// TIA Portal project "Factory_io_Analog_Assembler_with tia_portal_s7_plc1200_sequential" (V16)

(* hardware
DEVICE "S7-1200 station_1"  S7-1200 Station
   slot 0: "Rack_0"  S7-1200 Rack  Rack  V1.0
   slot 1: "PLC_1"  CPU 1212C DC/DC/Rly  6ES7 212-1HE40-0XB0  V4.4
   slot 2: "AI 4x16BIT_1"  SM 1231 AI4 x HF  6ES7 231-5ND32-0XB0  V2.0
   slot 3: "AQ 2x16BIT_1"  SM 1232 AQ2  6ES7 232-4HB32-0XB0  V2.1
*)

// ===== PLC "PLC_1"  CPU 1212C DC/DC/Rly =====

VAR_GLOBAL   // PLC tag table "Default tag table"
   "X_Current_Value" AT %ID1 : Real;
   "Z_Current_Value" AT %ID5 : Real;
   "Set_X" AT %QD30 : Real;
   "Set_Z" AT %QD34 : Real;
   "x scale for x" AT %MD44 : Real;
   "x rounded" AT %MD88 : Real;   // x rounded *10
   "Scale_X_For_Z" AT %MD48 : Real;
   "Z_rounded" AT %MD84 : Real;   // z rounded * 10
   "Item Detected" AT %I0.0 : Bool;
   "Lid At Place" AT %I0.1 : Bool;
   "Base At Place" AT %I0.2 : Bool;
   "Part Leaving" AT %I0.3 : Bool;
   "Start" AT %I0.4 : Bool;
   "Reset" AT %I0.5 : Bool;
   "Manual" AT %I0.6 : Bool;
   "auto" AT %I0.7 : Bool;
   "Lid Conveyor 1" AT %Q0.0 : Bool;
   "Stop Blade     1" AT %Q0.1 : Bool;
   "Lid Conveyor 2" AT %Q0.2 : Bool;
   "Base Conveyor 1" AT %Q0.3 : Bool;
   "Stop blad        2" AT %Q0.4 : Bool;
   "Base Conveyor 2" AT %Q0.5 : Bool;
   "Grab" AT %Q0.6 : Bool;
   "Start Light" AT %Q0.7 : Bool;
   "Memory for Postive edge of start" AT %M0.0 : Bool;
   "Start_FC_one_time" AT %M0.1 : Bool;
   "Cycle complete" AT %M0.2 : Bool;
   "Negative edge for lid conveyor 1" AT %M0.3 : Bool;
   "Negative edge for base conveyor 1" AT %M0.4 : Bool;
   "Negative edge for grab" AT %M0.5 : Bool;
   "Negative edge for Stop Blade 2" AT %M0.6 : Bool;
   "Postive edge for lid at place" AT %M0.7 : Bool;
   "Postive Edge For Base At Place" AT %M1.0 : Bool;
   "Negative edge for part leaving" AT %M1.1 : Bool;
   "postive edge for part leaving" AT %M1.2 : Bool;
   "finished product counter" AT %QD38 : DWord;
END_VAR

DATA_BLOCK "modes"   // DB1
{ S7_Optimized_Access := 'FALSE' }
VERSION : 0.1
   VAR
      "Reset Mode" : Bool;
      "Manual Mode" : Bool;
      "Auto Mode" : Bool;
   END_VAR
BEGIN
END_DATA_BLOCK

DATA_BLOCK "Step_Data"   // DB2
{ S7_Optimized_Access := 'TRUE' }
VERSION : 0.1
   VAR
      "Set X" : Real;
      "Set Z" : Real;
      "Lid Conveyor 1" : Bool;
      "Base Conveyor 1" : Bool;
      "Base Conveyor 2" : Bool;
      Grab : Bool;
      "Stop Blade 1" : Bool;
      "Stop Blade 2" : Bool;
      Every_thing_AT_home : Bool;
   END_VAR
BEGIN
END_DATA_BLOCK

DATA_BLOCK "Steps"   // DB3
{ S7_Optimized_Access := 'TRUE' }
VERSION : 0.1
   VAR
      Current_step : Int;
   END_VAR
BEGIN
END_DATA_BLOCK

// folder: System blocks/Program resources

DATA_BLOCK "IEC_Counter_0_DB"   // DB4
{ S7_Optimized_Access := 'TRUE' }
AUTHOR : Simatic
FAMILY : IEC
NAME : CNTR
VERSION : 1.0
// stored: InstanceOfName IEC_COUNTER
"IEC_COUNTER"
BEGIN
END_DATA_BLOCK

// folder: (top level)

FUNCTION "round_x and z" : Void   // FC1, LAD
{ S7_Optimized_Access := 'TRUE' }
VERSION : 0.1
BEGIN

REGION Network 1
   // Z rounded x10
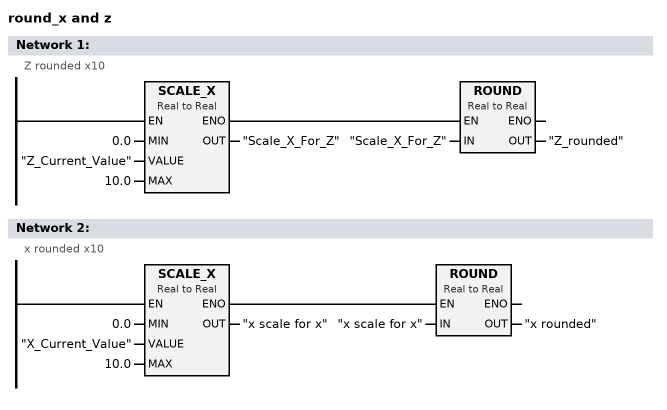
   RUNG wire#powerrail
      { S7_Templates := "[SrcType := Real, DestType := Real]" } Scale(min := 0.0, value := "Z_Current_Value", max := 10.0, out => "Scale_X_For_Z")
      { S7_Templates := "[SrcType := Real, DestType := Real]" } Round(in := "Scale_X_For_Z", out => "Z_rounded")
   END_RUNG
   // the same network as SCL:
   "Scale_X_For_Z" := SCALE_X(MIN := 0.0, VALUE := "Z_Current_Value", MAX := 10.0);
   "Z_rounded" := ROUND("Scale_X_For_Z");
END_REGION

REGION Network 2
   // x rounded x10
   RUNG wire#powerrail
      { S7_Templates := "[SrcType := Real, DestType := Real]" } Scale(min := 0.0, value := "X_Current_Value", max := 10.0, out => "x scale for x")
      { S7_Templates := "[SrcType := Real, DestType := Real]" } Round(in := "x scale for x", out => "x rounded")
   END_RUNG
   // the same network as SCL:
   "x scale for x" := SCALE_X(MIN := 0.0, VALUE := "X_Current_Value", MAX := 10.0);
   "x rounded" := ROUND("x scale for x");
END_REGION
END_FUNCTION

FUNCTION "Step_definition" : Void   // FC2, LAD
{ S7_Optimized_Access := 'TRUE' }
VERSION : 0.1
   VAR_TEMP   // added for the SCL form of the ladder/FBD networks
      _w1 : Bool;
   END_VAR
BEGIN

REGION Network 1: turn on lid conveyor till lid at place
   // start pressed  and every thing at home
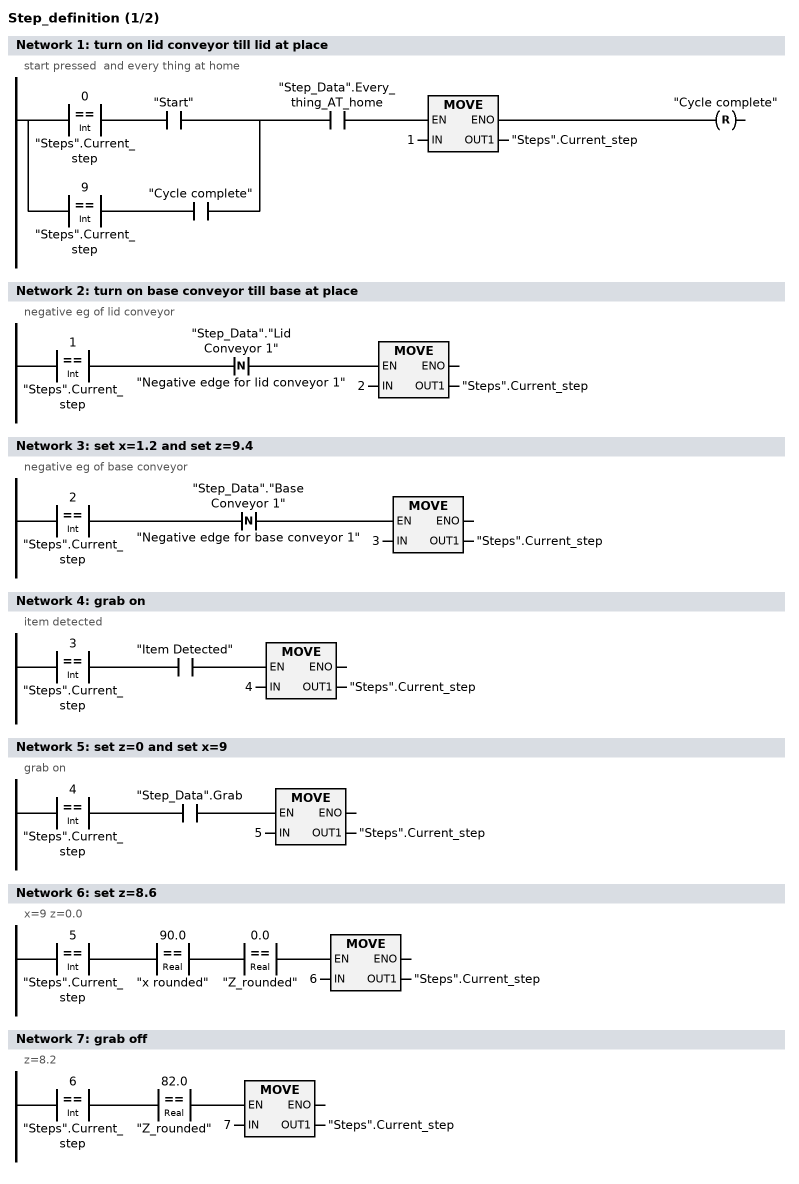
   RUNG wire#powerrail
      { S7_Templates := "SrcType := Int" } EQ_Contact(in1 := 0, in2 := "Steps".Current_step)
      Contact( "Start" )
      wire#w1
      Contact( "Step_Data".Every_thing_AT_home )
      Move(in := 1, out1 => "Steps".Current_step)
      R_Coil( "Cycle complete" )
   END_RUNG
   RUNG wire#powerrail
      { S7_Templates := "SrcType := Int" } EQ_Contact(in1 := 9, in2 := "Steps".Current_step)
      Contact( "Cycle complete" )
   END_RUNG wire#w1
   // the same network as SCL:
   #_w1 := (((0 = "Steps".Current_step) AND "Start") OR ((9 = "Steps".Current_step) AND "Cycle complete")) AND "Step_Data".Every_thing_AT_home;
   IF #_w1 THEN
       "Steps".Current_step := 1;
       "Cycle complete" := FALSE;
   END_IF;
END_REGION

REGION Network 2: turn on base conveyor till base at place
   // negative eg of lid conveyor
   RUNG wire#powerrail
      { S7_Templates := "SrcType := Int" } EQ_Contact(in1 := 1, in2 := "Steps".Current_step)
      N_Contact(operand := "Step_Data"."Lid Conveyor 1", bit := "Negative edge for lid conveyor 1")
      Move(in := 2, out1 => "Steps".Current_step)
   END_RUNG
   // the same network as SCL:
   #_w1 := (1 = "Steps".Current_step) AND NOT "Step_Data"."Lid Conveyor 1" AND "Negative edge for lid conveyor 1";   // falling edge of "Step_Data"."Lid Conveyor 1"
   "Negative edge for lid conveyor 1" := "Step_Data"."Lid Conveyor 1";
   IF #_w1 THEN "Steps".Current_step := 2; END_IF;
END_REGION

REGION Network 3: set x=1.2 and set z=9.4
   // negative eg of base conveyor
   RUNG wire#powerrail
      { S7_Templates := "SrcType := Int" } EQ_Contact(in1 := 2, in2 := "Steps".Current_step)
      N_Contact(operand := "Step_Data"."Base Conveyor 1", bit := "Negative edge for base conveyor 1")
      Move(in := 3, out1 => "Steps".Current_step)
   END_RUNG
   // the same network as SCL:
   #_w1 := (2 = "Steps".Current_step) AND NOT "Step_Data"."Base Conveyor 1" AND "Negative edge for base conveyor 1";   // falling edge of "Step_Data"."Base Conveyor 1"
   "Negative edge for base conveyor 1" := "Step_Data"."Base Conveyor 1";
   IF #_w1 THEN "Steps".Current_step := 3; END_IF;
END_REGION

REGION Network 4: grab on
   // item detected
   RUNG wire#powerrail
      { S7_Templates := "SrcType := Int" } EQ_Contact(in1 := 3, in2 := "Steps".Current_step)
      Contact( "Item Detected" )
      Move(in := 4, out1 => "Steps".Current_step)
   END_RUNG
   // the same network as SCL:
   IF (3 = "Steps".Current_step) AND "Item Detected" THEN "Steps".Current_step := 4; END_IF;
END_REGION

REGION Network 5: set z=0 and set x=9
   // grab on
   RUNG wire#powerrail
      { S7_Templates := "SrcType := Int" } EQ_Contact(in1 := 4, in2 := "Steps".Current_step)
      Contact( "Step_Data".Grab )
      Move(in := 5, out1 => "Steps".Current_step)
   END_RUNG
   // the same network as SCL:
   IF (4 = "Steps".Current_step) AND "Step_Data".Grab THEN "Steps".Current_step := 5; END_IF;
END_REGION

REGION Network 6: set z=8.6
   // x=9 z=0.0
   RUNG wire#powerrail
      { S7_Templates := "SrcType := Int" } EQ_Contact(in1 := 5, in2 := "Steps".Current_step)
      { S7_Templates := "SrcType := Real" } EQ_Contact(in1 := 90.0, in2 := "x rounded")
      { S7_Templates := "SrcType := Real" } EQ_Contact(in1 := 0.0, in2 := "Z_rounded")
      Move(in := 6, out1 => "Steps".Current_step)
   END_RUNG
   // the same network as SCL:
   IF (5 = "Steps".Current_step) AND (90.0 = "x rounded") AND (0.0 = "Z_rounded") THEN
       "Steps".Current_step := 6;
   END_IF;
END_REGION

REGION Network 7: grab off
   // z=8.2
   RUNG wire#powerrail
      { S7_Templates := "SrcType := Int" } EQ_Contact(in1 := 6, in2 := "Steps".Current_step)
      { S7_Templates := "SrcType := Real" } EQ_Contact(in1 := 82.0, in2 := "Z_rounded")
      Move(in := 7, out1 => "Steps".Current_step)
   END_RUNG
   // the same network as SCL:
   IF (6 = "Steps".Current_step) AND (82.0 = "Z_rounded") THEN "Steps".Current_step := 7; END_IF;
END_REGION

REGION Network 8: stop blade2 off
   // negative eg of grab
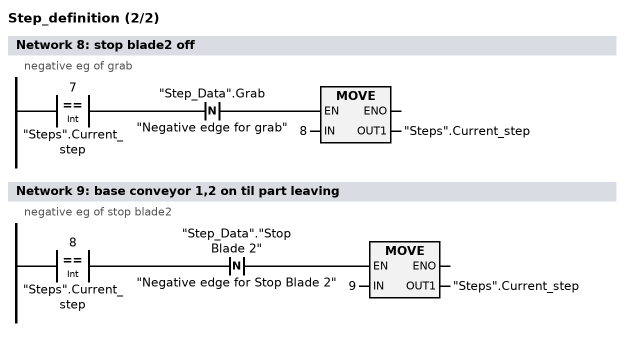
   RUNG wire#powerrail
      { S7_Templates := "SrcType := Int" } EQ_Contact(in1 := 7, in2 := "Steps".Current_step)
      N_Contact(operand := "Step_Data".Grab, bit := "Negative edge for grab")
      Move(in := 8, out1 => "Steps".Current_step)
   END_RUNG
   // the same network as SCL:
   #_w1 := (7 = "Steps".Current_step) AND NOT "Step_Data".Grab AND "Negative edge for grab";   // falling edge of "Step_Data".Grab
   "Negative edge for grab" := "Step_Data".Grab;
   IF #_w1 THEN "Steps".Current_step := 8; END_IF;
END_REGION

REGION Network 9: base conveyor 1,2 on til part leaving
   // negative eg of stop blade2
   RUNG wire#powerrail
      { S7_Templates := "SrcType := Int" } EQ_Contact(in1 := 8, in2 := "Steps".Current_step)
      N_Contact(operand := "Step_Data"."Stop Blade 2", bit := "Negative edge for Stop Blade 2")
      Move(in := 9, out1 => "Steps".Current_step)
   END_RUNG
   // the same network as SCL:
   #_w1 := (8 = "Steps".Current_step) AND NOT "Step_Data"."Stop Blade 2" AND "Negative edge for Stop Blade 2";   // falling edge of "Step_Data"."Stop Blade 2"
   "Negative edge for Stop Blade 2" := "Step_Data"."Stop Blade 2";
   IF #_w1 THEN "Steps".Current_step := 9; END_IF;
END_REGION
END_FUNCTION

FUNCTION "Step_Execution" : Void   // FC3, LAD
{ S7_Optimized_Access := 'TRUE' }
VERSION : 0.1
   VAR_TEMP   // added for the SCL form of the ladder/FBD networks
      _w1 : Bool;
      _w2 : Bool;
      _w3 : Bool;
   END_VAR
BEGIN

REGION Network 1: turn on lid conveyor till lid at place
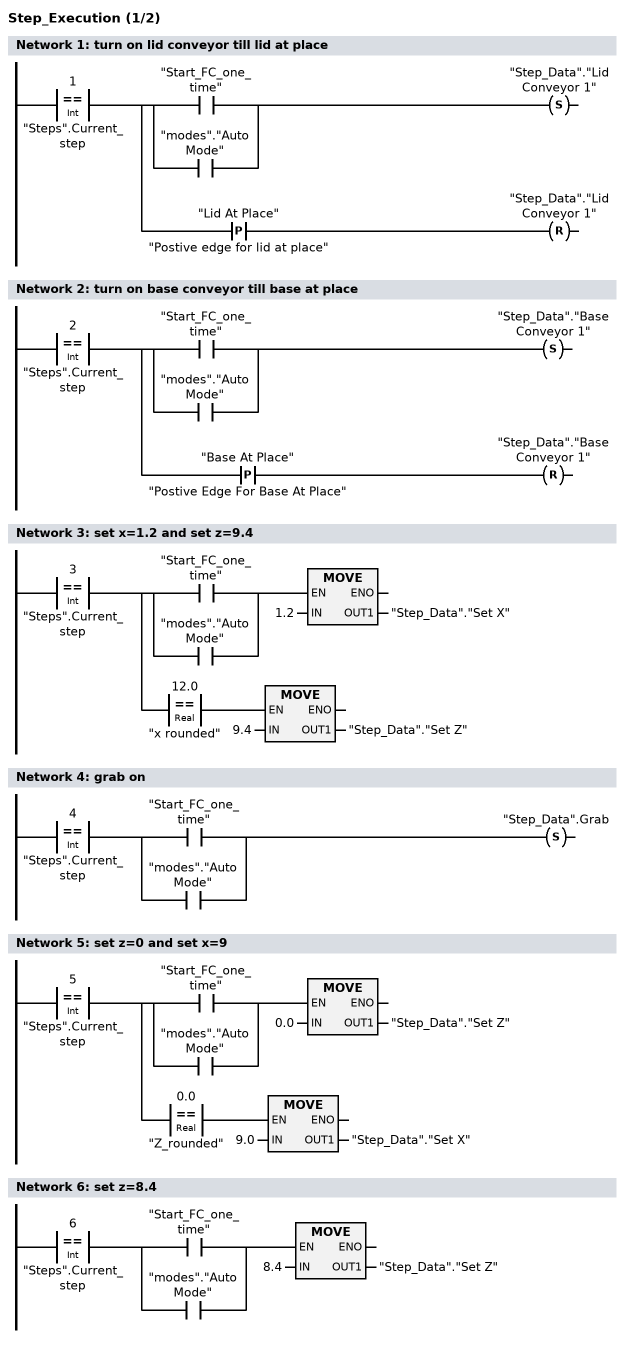
   RUNG wire#powerrail
      { S7_Templates := "SrcType := Int" } EQ_Contact(in1 := 1, in2 := "Steps".Current_step)
      wire#w1
      Contact( "Start_FC_one_time" )
      wire#w2
      S_Coil( "Step_Data"."Lid Conveyor 1" )
   END_RUNG
   RUNG wire#w1
      Contact( "modes"."Auto Mode" )
   END_RUNG wire#w2
   RUNG wire#w1
      P_Contact(operand := "Lid At Place", bit := "Postive edge for lid at place")
      R_Coil( "Step_Data"."Lid Conveyor 1" )
   END_RUNG
   // the same network as SCL:
   #_w1 := 1 = "Steps".Current_step;
   IF #_w1 AND ("Start_FC_one_time" OR "modes"."Auto Mode") THEN
       "Step_Data"."Lid Conveyor 1" := TRUE;
   END_IF;
   #_w2 := #_w1 AND "Lid At Place" AND NOT "Postive edge for lid at place";   // rising edge of "Lid At Place"
   "Postive edge for lid at place" := "Lid At Place";
   IF #_w2 THEN "Step_Data"."Lid Conveyor 1" := FALSE; END_IF;
END_REGION

REGION Network 2: turn on base conveyor till base at place
   RUNG wire#powerrail
      { S7_Templates := "SrcType := Int" } EQ_Contact(in1 := 2, in2 := "Steps".Current_step)
      wire#w1
      Contact( "Start_FC_one_time" )
      wire#w2
      S_Coil( "Step_Data"."Base Conveyor 1" )
   END_RUNG
   RUNG wire#w1
      Contact( "modes"."Auto Mode" )
   END_RUNG wire#w2
   RUNG wire#w1
      P_Contact(operand := "Base At Place", bit := "Postive Edge For Base At Place")
      R_Coil( "Step_Data"."Base Conveyor 1" )
   END_RUNG
   // the same network as SCL:
   #_w1 := 2 = "Steps".Current_step;
   IF #_w1 AND ("Start_FC_one_time" OR "modes"."Auto Mode") THEN
       "Step_Data"."Base Conveyor 1" := TRUE;
   END_IF;
   #_w2 := #_w1 AND "Base At Place" AND NOT "Postive Edge For Base At Place";   // rising edge of "Base At Place"
   "Postive Edge For Base At Place" := "Base At Place";
   IF #_w2 THEN "Step_Data"."Base Conveyor 1" := FALSE; END_IF;
END_REGION

REGION Network 3: set x=1.2 and set z=9.4
   RUNG wire#powerrail
      { S7_Templates := "SrcType := Int" } EQ_Contact(in1 := 3, in2 := "Steps".Current_step)
      wire#w1
      Contact( "Start_FC_one_time" )
      wire#w2
      Move(in := 1.2, out1 => "Step_Data"."Set X")
   END_RUNG
   RUNG wire#w1
      Contact( "modes"."Auto Mode" )
   END_RUNG wire#w2
   RUNG wire#w1
      { S7_Templates := "SrcType := Real" } EQ_Contact(in1 := 12.0, in2 := "x rounded")
      Move(in := 9.4, out1 => "Step_Data"."Set Z")
   END_RUNG
   // the same network as SCL:
   #_w1 := 3 = "Steps".Current_step;
   IF #_w1 AND ("Start_FC_one_time" OR "modes"."Auto Mode") THEN "Step_Data"."Set X" := 1.2; END_IF;
   IF #_w1 AND (12.0 = "x rounded") THEN "Step_Data"."Set Z" := 9.4; END_IF;
END_REGION

REGION Network 4: grab on
   RUNG wire#powerrail
      { S7_Templates := "SrcType := Int" } EQ_Contact(in1 := 4, in2 := "Steps".Current_step)
      wire#w1
      Contact( "Start_FC_one_time" )
      wire#w2
      S_Coil( "Step_Data".Grab )
   END_RUNG
   RUNG wire#w1
      Contact( "modes"."Auto Mode" )
   END_RUNG wire#w2
   // the same network as SCL:
   IF (4 = "Steps".Current_step) AND ("Start_FC_one_time" OR "modes"."Auto Mode") THEN
       "Step_Data".Grab := TRUE;
   END_IF;
END_REGION

REGION Network 5: set z=0 and set x=9
   RUNG wire#powerrail
      { S7_Templates := "SrcType := Int" } EQ_Contact(in1 := 5, in2 := "Steps".Current_step)
      wire#w1
      Contact( "Start_FC_one_time" )
      wire#w2
      Move(in := 0.0, out1 => "Step_Data"."Set Z")
   END_RUNG
   RUNG wire#w1
      Contact( "modes"."Auto Mode" )
   END_RUNG wire#w2
   RUNG wire#w1
      { S7_Templates := "SrcType := Real" } EQ_Contact(in1 := 0.0, in2 := "Z_rounded")
      Move(in := 9.0, out1 => "Step_Data"."Set X")
   END_RUNG
   // the same network as SCL:
   #_w1 := 5 = "Steps".Current_step;
   IF #_w1 AND ("Start_FC_one_time" OR "modes"."Auto Mode") THEN "Step_Data"."Set Z" := 0.0; END_IF;
   IF #_w1 AND (0.0 = "Z_rounded") THEN "Step_Data"."Set X" := 9.0; END_IF;
END_REGION

REGION Network 6: set z=8.4
   RUNG wire#powerrail
      { S7_Templates := "SrcType := Int" } EQ_Contact(in1 := 6, in2 := "Steps".Current_step)
      wire#w1
      Contact( "Start_FC_one_time" )
      wire#w2
      Move(in := 8.4, out1 => "Step_Data"."Set Z")
   END_RUNG
   RUNG wire#w1
      Contact( "modes"."Auto Mode" )
   END_RUNG wire#w2
   // the same network as SCL:
   IF (6 = "Steps".Current_step) AND ("Start_FC_one_time" OR "modes"."Auto Mode") THEN
       "Step_Data"."Set Z" := 8.4;
   END_IF;
END_REGION

REGION Network 7: grab off
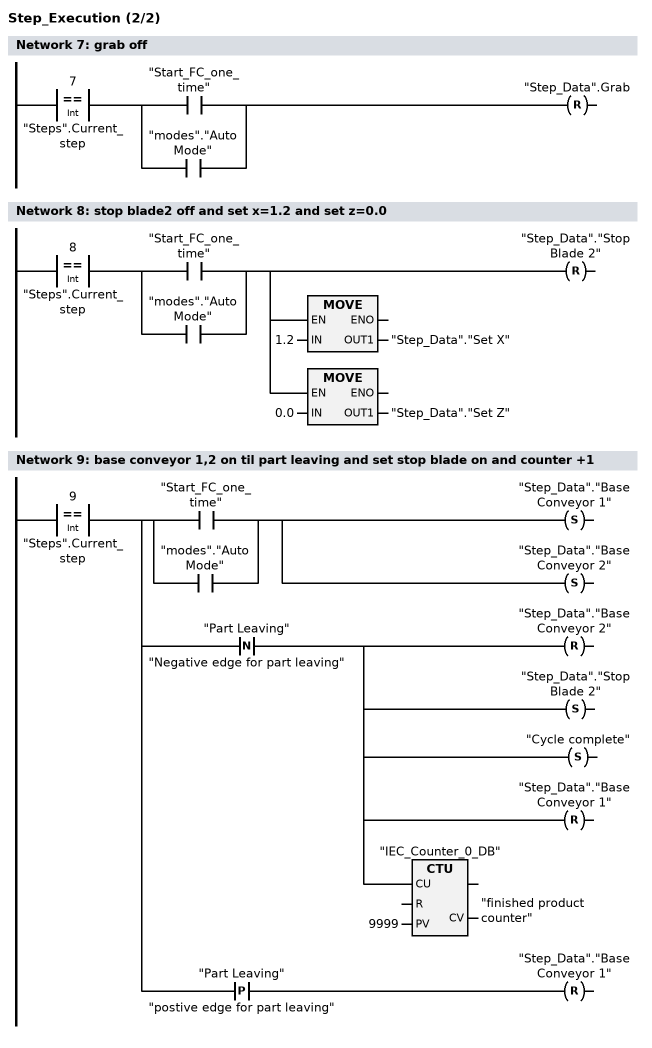
   RUNG wire#powerrail
      { S7_Templates := "SrcType := Int" } EQ_Contact(in1 := 7, in2 := "Steps".Current_step)
      wire#w1
      Contact( "Start_FC_one_time" )
      wire#w2
      R_Coil( "Step_Data".Grab )
   END_RUNG
   RUNG wire#w1
      Contact( "modes"."Auto Mode" )
   END_RUNG wire#w2
   // the same network as SCL:
   IF (7 = "Steps".Current_step) AND ("Start_FC_one_time" OR "modes"."Auto Mode") THEN
       "Step_Data".Grab := FALSE;
   END_IF;
END_REGION

REGION Network 8: stop blade2 off and set x=1.2 and set z=0.0
   RUNG wire#powerrail
      { S7_Templates := "SrcType := Int" } EQ_Contact(in1 := 8, in2 := "Steps".Current_step)
      wire#w1
      Contact( "Start_FC_one_time" )
      wire#w2
      R_Coil( "Step_Data"."Stop Blade 2" )
   END_RUNG
   RUNG wire#w1
      Contact( "modes"."Auto Mode" )
   END_RUNG wire#w2
   RUNG wire#w2
      Move(in := 1.2, out1 => "Step_Data"."Set X")
   END_RUNG
   RUNG wire#w2
      Move(in := 0.0, out1 => "Step_Data"."Set Z")
   END_RUNG
   // the same network as SCL:
   IF (8 = "Steps".Current_step) AND ("Start_FC_one_time" OR "modes"."Auto Mode") THEN
       "Step_Data"."Stop Blade 2" := FALSE;
       "Step_Data"."Set X" := 1.2;
       "Step_Data"."Set Z" := 0.0;
   END_IF;
END_REGION

REGION Network 9: base conveyor 1,2 on til part leaving and set stop blade on and counter +1
   #_w1 := 9 = "Steps".Current_step;
   IF #_w1 AND ("Start_FC_one_time" OR "modes"."Auto Mode") THEN
       "Step_Data"."Base Conveyor 1" := TRUE;
       "Step_Data"."Base Conveyor 2" := TRUE;
   END_IF;
   #_w2 := #_w1 AND NOT "Part Leaving" AND "Negative edge for part leaving";   // falling edge of "Part Leaving"
   "Negative edge for part leaving" := "Part Leaving";
   IF #_w2 THEN
       "Step_Data"."Base Conveyor 2" := FALSE;
       "Step_Data"."Stop Blade 2" := TRUE;
       "Cycle complete" := TRUE;
       "Step_Data"."Base Conveyor 1" := FALSE;
   END_IF;
   "IEC_Counter_0_DB".CTU(CU := #_w2, PV := 9999, CV => "finished product counter");
   #_w3 := #_w1 AND "Part Leaving" AND NOT "postive edge for part leaving";   // rising edge of "Part Leaving"
   "postive edge for part leaving" := "Part Leaving";
   IF #_w3 THEN "Step_Data"."Base Conveyor 1" := FALSE; END_IF;
END_REGION
END_FUNCTION

FUNCTION "Assignment" : Void   // FC4, LAD
{ S7_Optimized_Access := 'TRUE' }
VERSION : 0.1
BEGIN

REGION Network 1
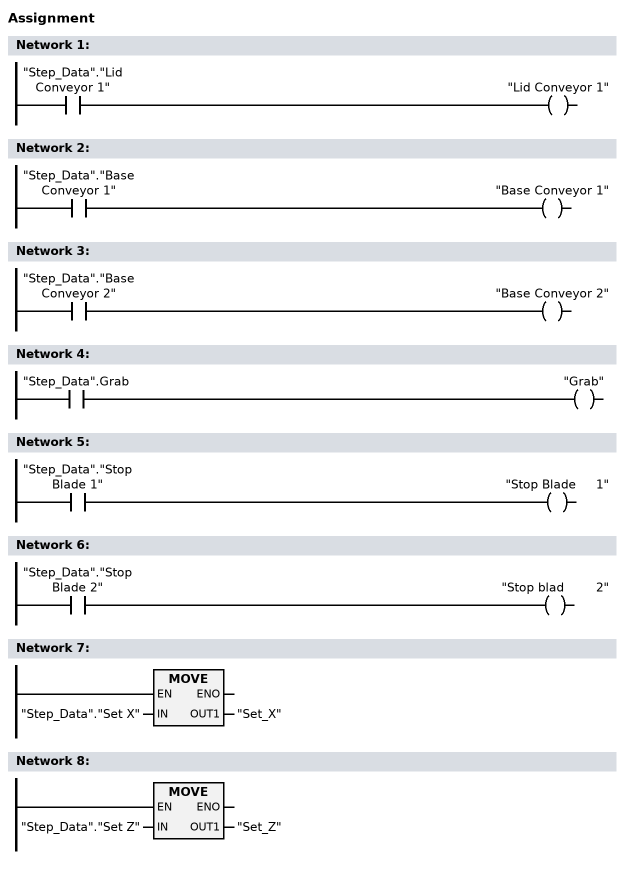
   RUNG wire#powerrail
      Contact( "Step_Data"."Lid Conveyor 1" )
      Coil( "Lid Conveyor 1" )
   END_RUNG
   // the same network as SCL:
   "Lid Conveyor 1" := "Step_Data"."Lid Conveyor 1";
END_REGION

REGION Network 2
   RUNG wire#powerrail
      Contact( "Step_Data"."Base Conveyor 1" )
      Coil( "Base Conveyor 1" )
   END_RUNG
   // the same network as SCL:
   "Base Conveyor 1" := "Step_Data"."Base Conveyor 1";
END_REGION

REGION Network 3
   RUNG wire#powerrail
      Contact( "Step_Data"."Base Conveyor 2" )
      Coil( "Base Conveyor 2" )
   END_RUNG
   // the same network as SCL:
   "Base Conveyor 2" := "Step_Data"."Base Conveyor 2";
END_REGION

REGION Network 4
   RUNG wire#powerrail
      Contact( "Step_Data".Grab )
      Coil( "Grab" )
   END_RUNG
   // the same network as SCL:
   "Grab" := "Step_Data".Grab;
END_REGION

REGION Network 5
   RUNG wire#powerrail
      Contact( "Step_Data"."Stop Blade 1" )
      Coil( "Stop Blade     1" )
   END_RUNG
   // the same network as SCL:
   "Stop Blade     1" := "Step_Data"."Stop Blade 1";
END_REGION

REGION Network 6
   RUNG wire#powerrail
      Contact( "Step_Data"."Stop Blade 2" )
      Coil( "Stop blad        2" )
   END_RUNG
   // the same network as SCL:
   "Stop blad        2" := "Step_Data"."Stop Blade 2";
END_REGION

REGION Network 7
   RUNG wire#powerrail
      Move(in := "Step_Data"."Set X", out1 => "Set_X")
   END_RUNG
   // the same network as SCL:
   "Set_X" := "Step_Data"."Set X";
END_REGION

REGION Network 8
   RUNG wire#powerrail
      Move(in := "Step_Data"."Set Z", out1 => "Set_Z")
   END_RUNG
   // the same network as SCL:
   "Set_Z" := "Step_Data"."Set Z";
END_REGION
END_FUNCTION

FUNCTION "Operating Mode" : Void   // FC5, LAD
{ S7_Optimized_Access := 'TRUE' }
VERSION : 0.1
   VAR_TEMP   // added for the SCL form of the ladder/FBD networks
      _w1 : Bool;
      _w2 : Bool;
   END_VAR
BEGIN

REGION Network 1
   // manual
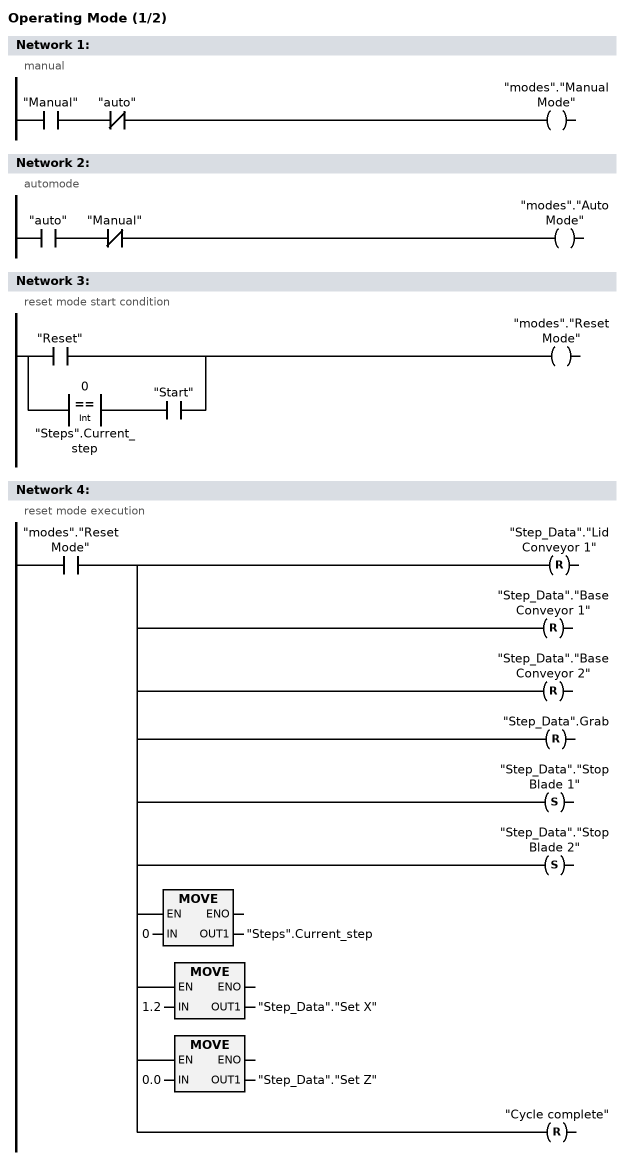
   RUNG wire#powerrail
      Contact( "Manual" )
      I_Contact( "auto" )
      Coil( "modes"."Manual Mode" )
   END_RUNG
   // the same network as SCL:
   "modes"."Manual Mode" := "Manual" AND NOT "auto";
END_REGION

REGION Network 2
   // automode
   RUNG wire#powerrail
      Contact( "auto" )
      I_Contact( "Manual" )
      Coil( "modes"."Auto Mode" )
   END_RUNG
   // the same network as SCL:
   "modes"."Auto Mode" := "auto" AND NOT "Manual";
END_REGION

REGION Network 3
   // reset mode start condition
   RUNG wire#powerrail
      Contact( "Reset" )
      wire#w1
      Coil( "modes"."Reset Mode" )
   END_RUNG
   RUNG wire#powerrail
      { S7_Templates := "SrcType := Int" } EQ_Contact(in1 := 0, in2 := "Steps".Current_step)
      Contact( "Start" )
   END_RUNG wire#w1
   // the same network as SCL:
   "modes"."Reset Mode" := "Reset" OR ((0 = "Steps".Current_step) AND "Start");
END_REGION

REGION Network 4
   // reset mode execution
   RUNG wire#powerrail
      Contact( "modes"."Reset Mode" )
      wire#w1
      R_Coil( "Step_Data"."Lid Conveyor 1" )
   END_RUNG
   RUNG wire#w1
      R_Coil( "Step_Data"."Base Conveyor 1" )
   END_RUNG
   RUNG wire#w1
      R_Coil( "Step_Data"."Base Conveyor 2" )
   END_RUNG
   RUNG wire#w1
      R_Coil( "Step_Data".Grab )
   END_RUNG
   RUNG wire#w1
      S_Coil( "Step_Data"."Stop Blade 1" )
   END_RUNG
   RUNG wire#w1
      S_Coil( "Step_Data"."Stop Blade 2" )
   END_RUNG
   RUNG wire#w1
      Move(in := 0, out1 => "Steps".Current_step)
   END_RUNG
   RUNG wire#w1
      Move(in := 1.2, out1 => "Step_Data"."Set X")
   END_RUNG
   RUNG wire#w1
      Move(in := 0.0, out1 => "Step_Data"."Set Z")
   END_RUNG
   RUNG wire#w1
      R_Coil( "Cycle complete" )
   END_RUNG
   // the same network as SCL:
   IF "modes"."Reset Mode" THEN
       "Step_Data"."Lid Conveyor 1" := FALSE;
       "Step_Data"."Base Conveyor 1" := FALSE;
       "Step_Data"."Base Conveyor 2" := FALSE;
       "Step_Data".Grab := FALSE;
       "Step_Data"."Stop Blade 1" := TRUE;
       "Step_Data"."Stop Blade 2" := TRUE;
       "Steps".Current_step := 0;
       "Step_Data"."Set X" := 1.2;
       "Step_Data"."Set Z" := 0.0;
       "Cycle complete" := FALSE;
   END_IF;
END_REGION

REGION Network 5
   // one step
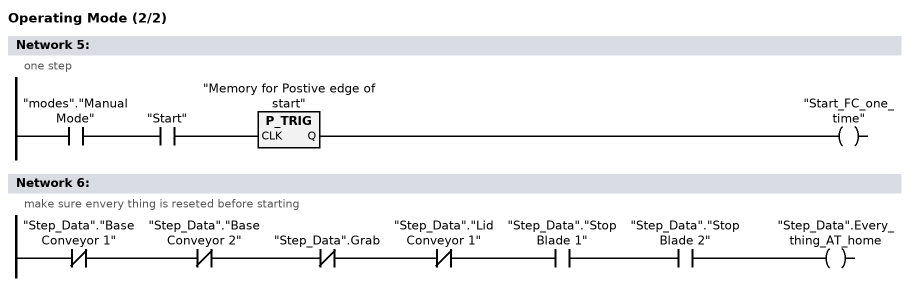
   RUNG wire#powerrail
      Contact( "modes"."Manual Mode" )
      Contact( "Start" )
      P_Trig( "Memory for Postive edge of start" )
      Coil( "Start_FC_one_time" )
   END_RUNG
   // the same network as SCL:
   #_w1 := "modes"."Manual Mode" AND "Start";
   #_w2 := #_w1 AND NOT "Memory for Postive edge of start";   // rising edge
   "Memory for Postive edge of start" := #_w1;
   "Start_FC_one_time" := #_w2;
END_REGION

REGION Network 6
   // make sure envery thing is reseted before starting
   RUNG wire#powerrail
      I_Contact( "Step_Data"."Base Conveyor 1" )
      I_Contact( "Step_Data"."Base Conveyor 2" )
      I_Contact( "Step_Data".Grab )
      I_Contact( "Step_Data"."Lid Conveyor 1" )
      Contact( "Step_Data"."Stop Blade 1" )
      Contact( "Step_Data"."Stop Blade 2" )
      Coil( "Step_Data".Every_thing_AT_home )
   END_RUNG
   // the same network as SCL:
   "Step_Data".Every_thing_AT_home := NOT "Step_Data"."Base Conveyor 1" AND NOT "Step_Data"."Base Conveyor 2" AND NOT "Step_Data".Grab AND NOT "Step_Data"."Lid Conveyor 1" AND "Step_Data"."Stop Blade 1" AND "Step_Data"."Stop Blade 2";
END_REGION
END_FUNCTION

FUNCTION "MHJ-PLC-Lab-Function-S71200" : Void   // FC9000, SCL
{ S7_Optimized_Access := 'TRUE' }
VERSION : 0.1
   VAR_TEMP
      rdTimeReturn : Int;
      outputTime : DTL;
      SyncVal : Byte;
      forVal : Int;
      forVal_2 : Int;
      Value : Byte;
   END_VAR
   VAR CONSTANT
      CompVal : Byte := 16#34;
      Value_01 : Byte := 16#11;
      Value_01_DW : DWord := 16#A165_D992;
      Value_02_DW : DWord := 16#58BE_4401;
   END_VAR
BEGIN

   #Value:=PEEK(area := 16#82,
        dbNumber := 0,
        byteOffset := 511);
   #Value := #Value + 1;

   POKE(area := 16#82,
        dbNumber := 0,
        byteOffset := 511,
        value := #Value);

   POKE(area:=16#81,
        dbNumber:=0,
        byteOffset:=1016,
        value:=#Value_01_DW);
   POKE(area := 16#81,
        dbNumber := 0,
        byteOffset := 1020,
        value := #Value_02_DW);

   POKE(area := 16#81,
        dbNumber := 0,
        byteOffset := 511,
        value := B#16#00);

   FOR #forVal := 0 TO 120 DO
       FOR #forVal_2:=0 TO 10 DO
           #rdTimeReturn:=RD_SYS_T(#outputTime);
           #rdTimeReturn := WR_SYS_T(#outputTime);
           #rdTimeReturn := RD_SYS_T(#outputTime);
           #rdTimeReturn := WR_SYS_T(#outputTime);
       END_FOR;
       #SyncVal:= PEEK(area := 16#81,
                      dbNumber := 0,
                      byteOffset := 511);
       IF #SyncVal = #CompVal THEN
          GOTO M_1;
       END_IF;
   END_FOR;
   RETURN;

   M_1:
   POKE(area := 16#81,
        dbNumber := 0,
        byteOffset := 511,
        value := B#16#0);
END_FUNCTION

ORGANIZATION_BLOCK "Main"   // OB1, LAD, ProgramCycle
TITLE = "Main Program Sweep (Cycle)"
{ S7_Optimized_Access := 'TRUE' }
VERSION : 0.1
   VAR_INPUT
      Initial_Call : Bool;   // Initial call of this OB
      Remanence : Bool;   // =True, if remanent data are available
   END_VAR
BEGIN

REGION Network 1
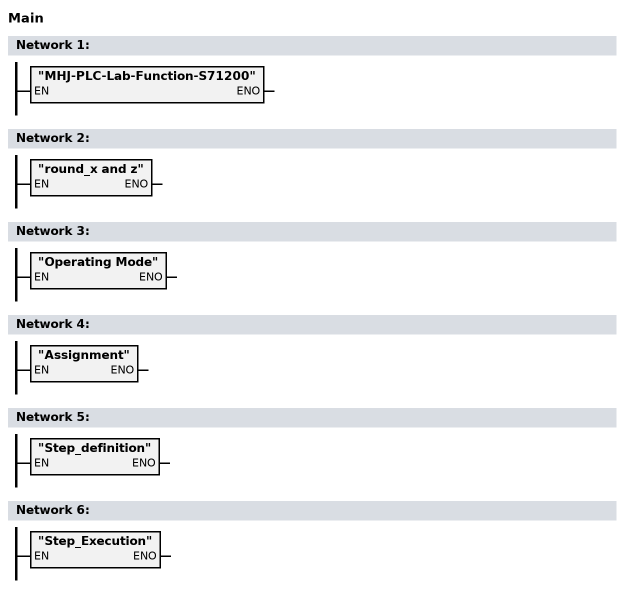
   RUNG wire#powerrail
      "MHJ-PLC-Lab-Function-S71200"()
   END_RUNG
   // the same network as SCL:
   "MHJ-PLC-Lab-Function-S71200"();
END_REGION

REGION Network 2
   RUNG wire#powerrail
      "round_x and z"()
   END_RUNG
   // the same network as SCL:
   "round_x and z"();
END_REGION

REGION Network 3
   RUNG wire#powerrail
      "Operating Mode"()
   END_RUNG
   // the same network as SCL:
   "Operating Mode"();
END_REGION

REGION Network 4
   RUNG wire#powerrail
      "Assignment"()
   END_RUNG
   // the same network as SCL:
   "Assignment"();
END_REGION

REGION Network 5
   RUNG wire#powerrail
      "Step_definition"()
   END_RUNG
   // the same network as SCL:
   "Step_definition"();
END_REGION

REGION Network 6
   RUNG wire#powerrail
      "Step_Execution"()
   END_RUNG
   // the same network as SCL:
   "Step_Execution"();
END_REGION
END_ORGANIZATION_BLOCK